# EPICS autosave request: iocBoot/obsolete/InstekPSP/auto_settings.req
file  "Omega_DP41_settings.req",         P=$(P), R=Omega1
